FUNCTION_BLOCK ABSTRACT AbstractReceiver IMPLEMENTS I_Callable, I_Receiver
VAR
	_tag: Tag;
END_VAR

(*
This method provides a standardized way for other objects to interact with the object that owns it.
*)
METHOD Call
VAR_INPUT
	iArg	: I_Arg;
END_VAR
END_METHOD

METHOD INTERNAL Receive
VAR_INPUT
	iArg			: I_Arg;
END_VAR
Call(iArg);
END_METHOD

(*
Provides access to the tag associated with the signal.
*)
PROPERTY FINAL Tag : I_Tag
GET
Tag := _tag;
END_GET
END_PROPERTY

END_FUNCTION_BLOCK

(* stored: Version 1.1.0.1
   POU AbstractReceiver: Id {21b26383-9808-407b-a8ba-abcd48a678b0}, SpecialFunc None
   Method Call: Id {a0f6c3b5-e234-4f8a-9a5e-368a72c8c866}
   Method Receive: Id {e0854879-c2ba-4c5c-b3ab-b6a2008b53db}
   Property Tag: Id {9ee99f7a-7a32-4794-966e-c9d5108d39b2}
   Get Get: Id {44574137-36bb-4b98-a702-3983fe897ba4} *)
